FUNCTION_BLOCK FB_Loader
VAR_INPUT
	EN : BOOL;
	Level_Prox : BOOL; // Loader Proximity Switch
	Flap_Reed : BOOL; // Loader Flap Reed Switch
	Switch : BOOL; // Loader switch
	PushButton : BOOL; // Loader Push Button
	Vac_Grant : BOOL; // Vacuum Grant to the Loader
	Switch_Bit : BOOL; // Loader internal Switch Bit - Push Button or Switch
END_VAR
VAR_OUTPUT
	ENO : BOOL;
	Valve : BOOL; // Loader Vacuum Valve
	Lamp : BOOL; // Loader status lamp
	Comp_Status : WORD; // Loader status word for Sysmetric Vision
	HMI_Status : WORD; // Loader status word for HMI
	Vac_Request : BOOL; // Vacuum Request from the loader
END_VAR
VAR
	Timer_0_1 : TON;		// 0.1 seconds timer for counters
	Timer0_5_s_ON : TON;	// 0.5 second TON for 1 second blink like P_1_0 from CJ
	Timer0_5_s_OFF : TOF;	// 0.5 second TOF for 1 second blink like P_1_0 from CJ
	Timer_50_ms_ON : TON;	// 50 mili second TON for 0.1 second blink like P_0_1 from CJ
	Timer_50_ms_OFF : TOF;	// 50 mili second TOF for 0.1 second blink like P_0_1 from CJ
	MATfallTIME : CTU;		// Material fall time after conveying usually 8 seconds
	Flap_Open_time : CTU;	// check if Flap is open for more than 1.5 second, if true cancel conveying alarm
	CONValarm : CTU;		// conveying alarm turn on after usually 4 bad conveyings
	One_Time : BOOL;		// allow a loader on dosing system to request conveying only one per vacuum grant from main PLC
	Switch_Keep : SR;		// Conveying Push botton switch
	Blink_1_0_s: BOOL;		// 1 second blink for loaders lamp when ON
	Blink_0_1_s: BOOL;		// 0.1 second blink for loaders lamp when alarm
END_VAR
VAR // added by the converter: edge detectors and wires of the graphical bodies
    _rt1, _rt2 : R_TRIG;
    _ft1 : F_TRIG;
    _w1, _w2, _w3 : BOOL;
END_VAR

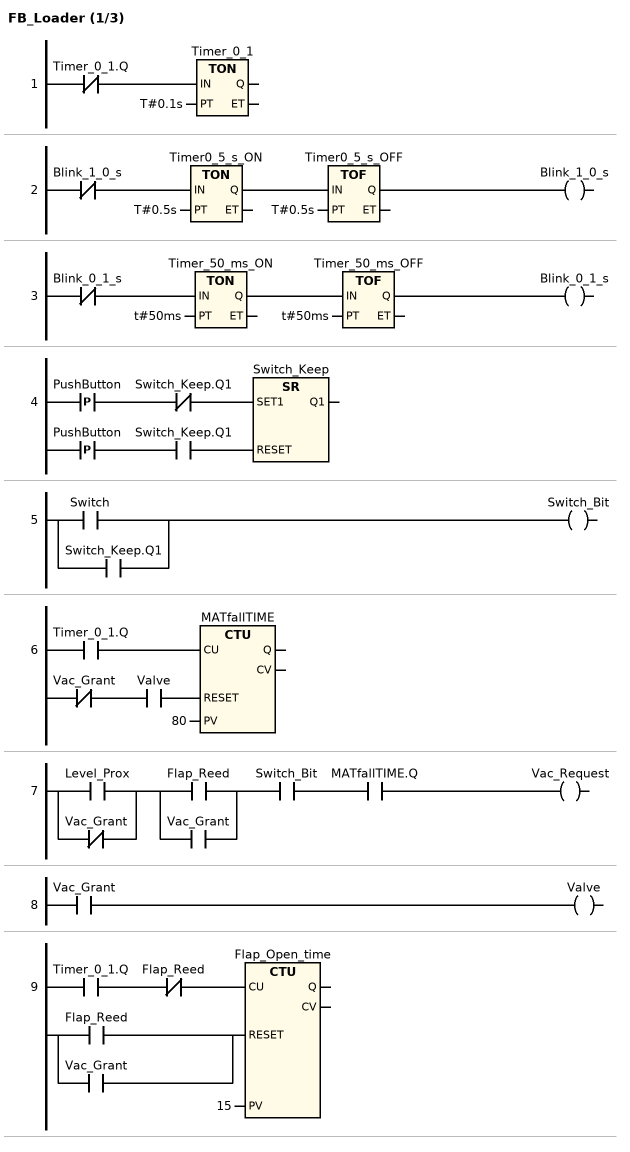
// NETWORK 1
Timer_0_1(IN := NOT Timer_0_1.Q, PT := T#0.1s); // TON

// NETWORK 2
Timer0_5_s_ON(IN := NOT Blink_1_0_s, PT := T#0.5s); // TON
Timer0_5_s_OFF(IN := Timer0_5_s_ON.Q, PT := T#0.5s); // TOF
Blink_1_0_s := Timer0_5_s_OFF.Q;

// NETWORK 3
Timer_50_ms_ON(IN := NOT Blink_0_1_s, PT := t#50ms); // TON
Timer_50_ms_OFF(IN := Timer_50_ms_ON.Q, PT := t#50ms); // TOF
Blink_0_1_s := Timer_50_ms_OFF.Q;

// NETWORK 4
_rt1(CLK := PushButton);
_rt2(CLK := PushButton);
Switch_Keep(SET1 := _rt1.Q AND NOT Switch_Keep.Q1, RESET := _rt2.Q AND Switch_Keep.Q1); // SR

// NETWORK 5
Switch_Bit := Switch OR Switch_Keep.Q1;

// NETWORK 6
MATfallTIME(CU := Timer_0_1.Q, RESET := NOT Vac_Grant AND Valve, PV := 80); // CTU

// NETWORK 7
Vac_Request := (Level_Prox OR NOT Vac_Grant) AND (Flap_Reed OR Vac_Grant) AND Switch_Bit AND MATfallTIME.Q;

// NETWORK 8
Valve := Vac_Grant;

// NETWORK 9
Flap_Open_time(CU := Timer_0_1.Q AND NOT Flap_Reed, RESET := Flap_Reed OR Vac_Grant, PV := 15); // CTU

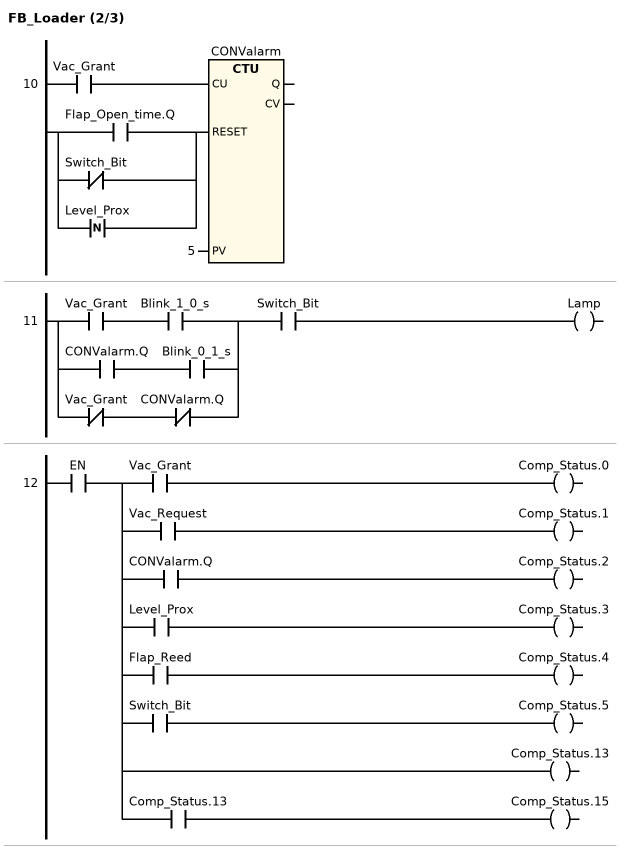
// NETWORK 10
_ft1(CLK := Level_Prox);
CONValarm(CU := Vac_Grant, RESET := Flap_Open_time.Q OR NOT Switch_Bit OR _ft1.Q, PV := 5); // CTU

// NETWORK 11
Lamp := (Vac_Grant AND Blink_1_0_s OR CONValarm.Q AND Blink_0_1_s OR NOT Vac_Grant AND NOT CONValarm.Q) AND Switch_Bit;

// NETWORK 12
Comp_Status.0 := EN AND Vac_Grant;
Comp_Status.1 := EN AND Vac_Request;
Comp_Status.2 := EN AND CONValarm.Q;
Comp_Status.3 := EN AND Level_Prox;
Comp_Status.4 := EN AND Flap_Reed;
Comp_Status.5 := EN AND Switch_Bit;
Comp_Status.13 := EN;
Comp_Status.15 := EN AND Comp_Status.13;

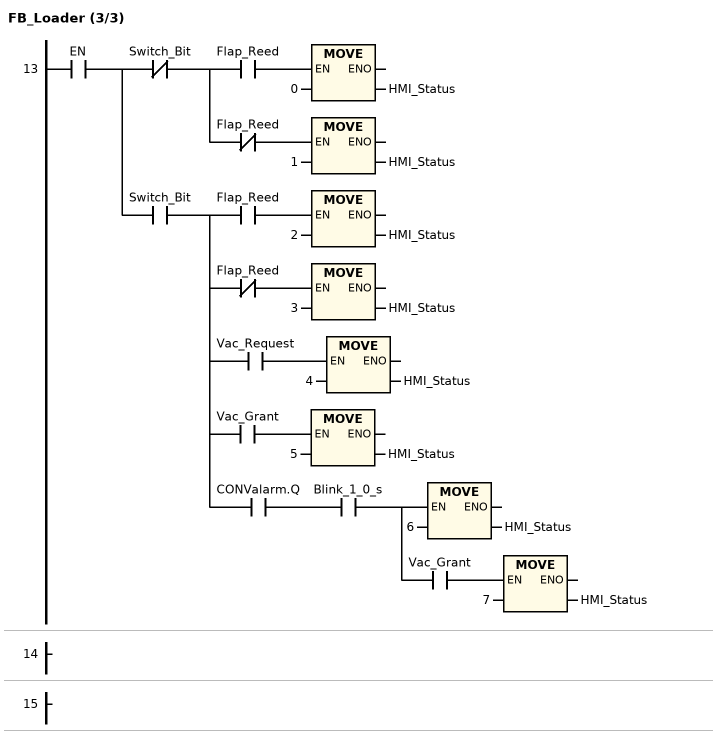
// NETWORK 13
_w1 := EN AND NOT Switch_Bit;
IF _w1 AND Flap_Reed THEN HMI_Status := 0; END_IF
IF _w1 AND NOT Flap_Reed THEN HMI_Status := 1; END_IF
_w2 := EN AND Switch_Bit;
IF _w2 AND Flap_Reed THEN HMI_Status := 2; END_IF
IF _w2 AND NOT Flap_Reed THEN HMI_Status := 3; END_IF
IF _w2 AND Vac_Request THEN HMI_Status := 4; END_IF
IF _w2 AND Vac_Grant THEN HMI_Status := 5; END_IF
_w3 := _w2 AND CONValarm.Q AND Blink_1_0_s;
IF _w3 THEN HMI_Status := 6; END_IF
IF _w3 AND Vac_Grant THEN HMI_Status := 7; END_IF

// NETWORK 14

// NETWORK 15

END_FUNCTION_BLOCK

(* stored: Version 1.1.0.1, ProductVersion 3.1.4024.13
   POU FB_Loader: Id {81e6a8e4-985e-48e1-92ce-6cdaa989c6d8}, SpecialFunc None *)
